TYPE ST_PCMStorageState :
STRUCT
	SOCValuePercentage : REAL; 
	SOCValueAbsolute : REAL; 
	TemperatureSensor : REAL; 
END_STRUCT
END_TYPE

(* stored: Version 1.1.0.1, ProductVersion 3.1.4024.10
   DUT ST_PCMStorageState: Id {783e6f4b-3647-4108-80c8-ea0c12c9f53c} *)
